FUNCTION_BLOCK FB_HEATING
VAR_INPUT
	ix_START: BOOL;
	TEMP: DINT;
	SETPOINT: DINT;
END_VAR
VAR_OUTPUT
	HEATING:BOOL;
END_VAR
VAR
	STATE: INT;
END_VAR

CASE STATE OF
	0: // Idle
        HEATING := FALSE;
        // Start cycle
        IF ix_START THEN
            STATE := 1;
        END_IF;
    1:
        IF ix_START = FALSE THEN
            STATE := 0;
        END_IF;
        IF (TEMP < SETPOINT) THEN
			HEATING :=TRUE;
		ELSE
			HEATING :=FALSE;
		END_IF
END_CASE;

END_FUNCTION_BLOCK

(* stored: Version 1.1.0.1, ProductVersion 3.1.4024.15
   POU FB_HEATING: Id {20d89b82-110c-46de-a9a3-a9f598c41c27}, SpecialFunc None *)
